(* PLC project Blank Project, Blank Blank 1.0 *)
(* stored: creationDateTime 2016-05-18T21:14:07, modificationDateTime 2023-04-28T12:49:40 *)

PROGRAM OverCurrent_XFMR2
  VAR
    Short_Circuit_XFMR2 : BOOL;
    Short_Circuit_66BUS2 : BOOL;
  END_VAR
  VAR
    Open_CB2_66KV AT %QX0.0 : BOOL;
    Open_CB3_66KV AT %QX0.1 : BOOL;
    Open_CB_XFMR2 AT %QX0.2 : BOOL;
    Open_CB2_22KV AT %QX0.3 : BOOL;
    Reset_All_CB AT %IX0.0 : BOOL;
    Current_CB2_66KV AT %IW0 : INT;
    Current_CB3_66KV AT %IW1 : INT;
    Current_XFMR2_W1 AT %IW2 : INT;
    Current_XFMR2_W2 AT %IW3 : INT;
    Current_CB_XFMR2 AT %IW4 : INT;
    Current_Fault_on_66BUS2 AT %IW5 : INT;
    Current_Fault_on_XFMR2 AT %IW6 : INT;
  END_VAR
  VAR CONSTANT
    Threshold : INT := 500;
  END_VAR

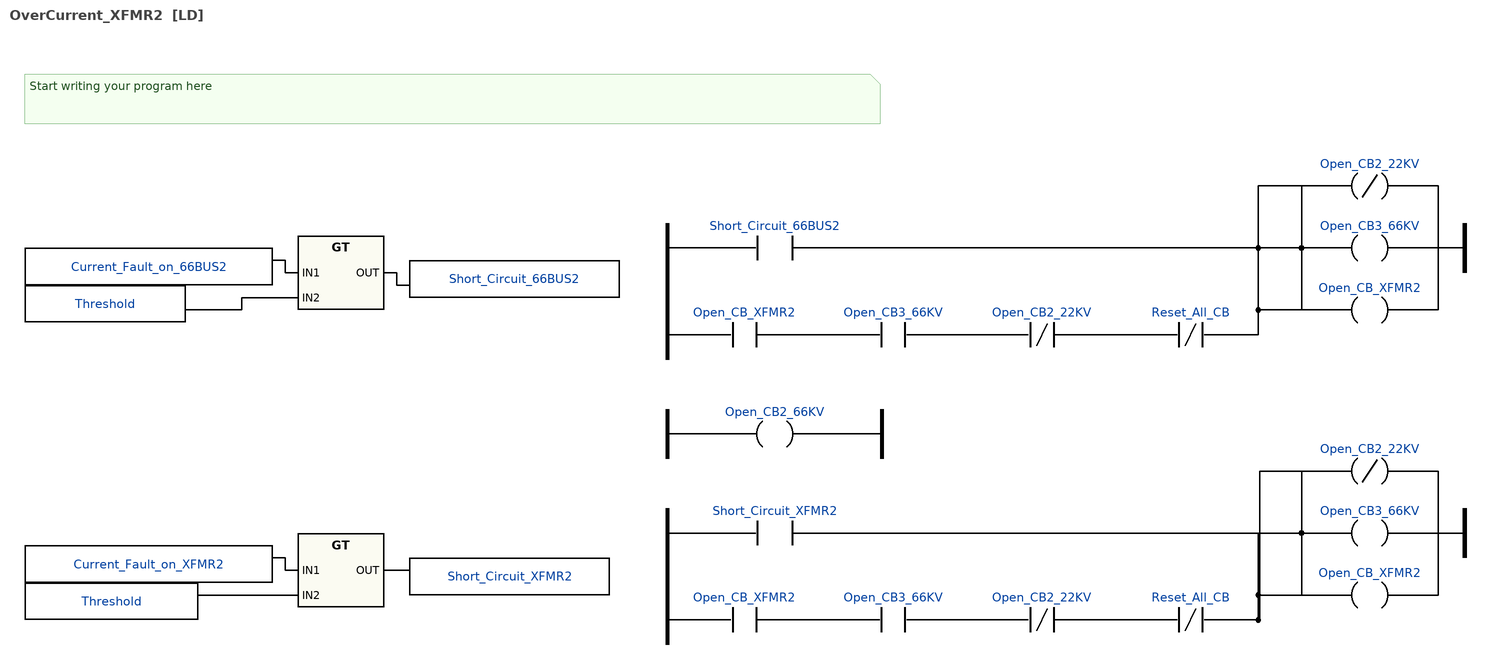
(* LD diagram, written out as Structured Text *)
(* Start writing your program here *)
Open_CB2_22KV := NOT (Short_Circuit_66BUS2 OR Open_CB_XFMR2 AND Open_CB3_66KV AND NOT Open_CB2_22KV AND NOT Reset_All_CB);
Open_CB3_66KV := Short_Circuit_66BUS2 OR Open_CB_XFMR2 AND Open_CB3_66KV AND NOT Open_CB2_22KV AND NOT Reset_All_CB;
Short_Circuit_66BUS2 := Current_Fault_on_66BUS2 > Threshold;
Open_CB_XFMR2 := Short_Circuit_66BUS2 OR Open_CB_XFMR2 AND Open_CB3_66KV AND NOT Open_CB2_22KV AND NOT Reset_All_CB;
Open_CB2_66KV := TRUE;
Open_CB2_22KV := NOT (Short_Circuit_XFMR2 OR Open_CB_XFMR2 AND Open_CB3_66KV AND NOT Open_CB2_22KV AND NOT Reset_All_CB);
Open_CB3_66KV := Short_Circuit_XFMR2 OR Open_CB_XFMR2 AND Open_CB3_66KV AND NOT Open_CB2_22KV AND NOT Reset_All_CB;
Short_Circuit_XFMR2 := Current_Fault_on_XFMR2 > Threshold;
Open_CB_XFMR2 := Short_Circuit_XFMR2 OR Open_CB_XFMR2 AND Open_CB3_66KV AND NOT Open_CB2_22KV AND NOT Reset_All_CB;
END_PROGRAM

CONFIGURATION Config0
  RESOURCE Res0 ON PLC
    TASK TaskMain(INTERVAL := T#10ms, PRIORITY := 0);
    PROGRAM Inst0 WITH TaskMain : OverCurrent_XFMR2;
  END_RESOURCE
END_CONFIGURATION
